# EPICS substitutions: epics/m-epics-TwinCATmotor/TwinCATmotorApp/Db/TwinCATmotor-extra.substitutions
file "TwinCATmotor-extra.template"
{
pattern
{P,      M,    R,   PORT, ADDR, HOMEPROC}
{IOC:,   m1, m1-,   MCU1,    1, 3       }
}
